{attribute addProperty BoxType "KL6841"}
{attribute addProperty Id "Channel_1Channel_1D2D48B900"}
{attribute addProperty CRC "996881571"}
{attribute addProperty SizeInBites "0"}
{attribute addProperty SizeInBytes "0"}
TYPE KL6841_3B6B34A3 :
STRUCT
	{attribute addProperty Name "Channel_1"}
	Channel_1 : Channel_1D2D48B9;
END_STRUCT
END_TYPE

(* stored: Version 1.2.0.0, ProductVersion 3.1.4024.9
   DUT KL6841_3B6B34A3: Id {d9a780b4-54e1-439e-b427-cd3eae44b608} *)
